TYPE ServicesTabs :
(
	OVERVIEW := 0,
    TIMING := 1,
    CONFIG := 2
);
END_TYPE

(* stored: Version 1.1.0.1, ProductVersion 3.1.4018.5
   DUT ServicesTabs: Id {605076d6-99e7-451f-af33-0e38d8c701a8} *)
